# EPICS autosave request: SCDLDApp/Db/dldDetectorv2_settings.req
$(P)$(R)ConfigFile
$(P)$(R)SizeT
$(P)$(R)MinTSI
$(P)$(R)SizeTSI
$(P)$(R)LiveImageXYAccum
$(P)$(R)TimeHistoAccum
$(P)$(R)H5EventsFilePath
$(P)$(R)H5EventsComment
file "ADBase_settings.req", P=$(P), R=$(R)
